	//外部输出端口Do对应的功能
	IF xSystemError OR xSystemWarning THEN
		DO_2:=FALSE;
	ELSE
		DO_2:=TRUE;
	END_IF
	DO_0:=xLED1Status;//设备运行指示灯	
	DO_1:=xLED2Status;//运行错误指示灯	
	//DO_2:= NOT xSystemError;// 机器人错误输出到外部设备
	//DO_4:=xAutoRun;//器人自动运行输出到外部设备
	
	IF CustomerPrgHandling.xWarning THEN//箱体越界信号
		WarningID:=30322;
	END_IF
	
	//////////////////////////////////////////////////////////////
	
	DeltaRobot_ErrorID:=Delta_Robot.eActiveErrorID;
	Xaxis_ErrorID	:=Axis_X.eActiveErrorID;
	Yaxis_ErrorID	:=Axis_Y.eActiveErrorID;
	Zaxis_ErrorID	:=Axis_Z.eActiveErrorID;
	A1axis_ErrorID  :=A1.eActiveErrorID;	
	A2axis_ErrorID	:=A2.eActiveErrorID;	
	A3axis_ErrorID	:=A3.eActiveErrorID;

	
	IF ErrorID<>0 THEN
		PrgOrParaErrorID:=ErrorID;
		ELSE
		PrgOrParaErrorID:=WarningID;
	END_IF

		//读取各轴的状态信息！
		ReadAxis1Info(Axis:=A1,Enable:=TRUE);
		ReadAxis2Info(Axis:=A2,Enable:=TRUE);
		ReadAxis3Info(Axis:=A3,Enable:=TRUE);

		
		//读取MCS坐标系下的位置	
		IF wstep<>20 THEN
		IF icschange=0 THEN
			AGBControl.eCoordSystem:=L_MC4P_CoordSystem.MCS;//笛卡尔坐标系MCS
			iCurrentCS:=L_MC4P_CoordSystem.MCS;
		END_IF
		IF icschange=1 THEN
			AGBControl.eCoordSystem:=L_MC4P_CoordSystem.ACS;//轴坐标系ACS
			iCurrentCS:=L_MC4P_CoordSystem.MCS;
		END_IF
		IF icschange=2 THEN
			AGBControl.eCoordSystem:=L_MC4P_CoordSystem.PCS_5;//PCS_5
			iCurrentCS:=L_MC4P_CoordSystem.PCS_5;
		END_IF
		IF icschange=4 THEN
			AGBControl.eCoordSystem:=L_MC4P_CoordSystem.PCS_6;//PCS_6
			iCurrentCS:=L_MC4P_CoordSystem.PCS_6;
		END_IF	
			ReadActPos_MCS.CoordSystem:=iCurrentCS;
			ReadActPos_MCS.Enable:=TRUE;
			ReadActPos_MCS(AxesGroup:=Delta_Robot);
			
			IF ReadActPos_MCS.Valid=TRUE THEN
				RobotPos.rRobotPosX:=LREAL_TO_REAL(ReadActPos_MCS.Position[1]);
				RobotPos.rRobotPosY:=LREAL_TO_REAL(ReadActPos_MCS.Position[2]);
				RobotPos.rRobotPosZ:=LREAL_TO_REAL(ReadActPos_MCS.Position[3]);
				
			END_IF
			
					
			ReadActPos_ACS.CoordSystem:=L_MC4P_CoordSystem.ACS;
			ReadActPos_ACS.Enable:=TRUE;
			ReadActPos_ACS(AxesGroup:=Delta_Robot);
			
			IF ReadActPos_ACS.Valid=TRUE THEN
				RobotPos.rRobotPosA1:=LREAL_TO_REAL(ReadActPos_ACS.Position[1]);
				RobotPos.rRobotPosA2:=LREAL_TO_REAL(ReadActPos_ACS.Position[2]);
				RobotPos.rRobotPosA3:=LREAL_TO_REAL(ReadActPos_ACS.Position[3]);
			END_IF
		END_IF
		
		Robot_Vel_X:=LREAL_TO_REAL(Delta_Robot.pAxis_X^.lrActVelocity);
		Robot_Vel_Y:=LREAL_TO_REAL(Delta_Robot.pAxis_Y^.lrActVelocity);
		Robot_Vel_Z:=LREAL_TO_REAL(Delta_Robot.pAxis_Z^.lrActVelocity);
		
		
		Robot_Vel_A1:=LREAL_TO_REAL(A1.lrActVelocity);
		Robot_Vel_A2:=LREAL_TO_REAL(A2.lrActVelocity);
		Robot_Vel_A3:=LREAL_TO_REAL(A3.lrActVelocity);
		//Infeed_Vel:=LREAL_TO_REAL(Infeeder.lrActVelocity);
		//Outfeed_Vel:=LREAL_TO_REAL(Outfeeder.lrActVelocity);
		//Infeed_Pos:=LREAL_TO_REAL(Infeeder.lrActPosition);
		//Outfeed_Pos:=LREAL_TO_REAL(Outfeeder.lrActPosition);
		//读取各轴的状态数据
		//读取X轴数据
		ReadXaxisPara[1].Enable:=TRUE;
		ReadXaxisPara[1].ParameterNumber:=51;
		rXaxis_PositiveLimit_Dsp:=LREAL_TO_REAL(ReadXaxisPara[1].Value);
		ReadXaxisPara[2].Enable:=TRUE;
		ReadXaxisPara[2].ParameterNumber:=52;
		rXaxis_NegativeLimit_Dsp:=LREAL_TO_REAL(ReadXaxisPara[2].Value);
		//读取Y轴数据
		ReadYaxisPara[1].Enable:=TRUE;
		ReadYaxisPara[1].ParameterNumber:=51;
		rYaxis_PositiveLimit_Dsp:=LREAL_TO_REAL(ReadYaxisPara[1].Value);
		ReadYaxisPara[2].Enable:=TRUE;
		ReadYaxisPara[2].ParameterNumber:=52;
		rYaxis_NegativeLimit_Dsp:=LREAL_TO_REAL(ReadYaxisPara[2].Value);
		//读取Z轴数据
		ReadZaxisPara[1].Enable:=TRUE;
		ReadZaxisPara[1].ParameterNumber:=51;
		rZaxis_PositiveLimit_Dsp:=LREAL_TO_REAL(ReadZaxisPara[1].Value);
		ReadZaxisPara[2].Enable:=TRUE;
		ReadZaxisPara[2].ParameterNumber:=52;
		rZaxis_NegativeLimit_Dsp:=LREAL_TO_REAL(ReadZaxisPara[2].Value);
		//读取A1轴数据
		CASE ReadA1_Step OF	
			0:
				ReadA1axisPara[1].ParameterNumber:=51;
				ReadA1axisPara[1].Enable:=TRUE;
				ReadA1_Step:=10;
			10:
				IF ReadA1axisPara[1].Valid AND NOT ReadA1axisPara[1].Error THEN
					rA1_PositiveLimit_Dsp:=LREAL_TO_REAL(ReadA1axisPara[1].Value);
					ReadA1axisPara[1].Enable:=FALSE;
					ReadA1_Step:=20;
				ELSE
					ReadA1_Step:=0;
				END_IF
			20:
				ReadA1axisPara[1].ParameterNumber:=52;
				ReadA1axisPara[1].Enable:=TRUE;
				ReadA1_Step:=30;
			30:
				IF ReadA1axisPara[1].Valid AND NOT ReadA1axisPara[1].Error THEN
					rA1_NegativeLimit_Dsp:=LREAL_TO_REAL(ReadA1axisPara[1].Value);
					ReadA1axisPara[1].Enable:=FALSE;
					ReadA1_Step:=40;
				ELSE
					ReadA1_Step:=20;
				END_IF
			40:
				ReadA1axisPara[1].ParameterNumber:=L_MC1P_IndexToParameter(16#2900,1,4);
				ReadA1axisPara[1].Enable:=TRUE;
				ReadA1_Step:=50;				
			50:
				IF ReadA1axisPara[1].Valid AND NOT ReadA1axisPara[1].Error THEN
					rA1_Vel_P1_Dsp:=LREAL_TO_REAL(ReadA1axisPara[1].Value/100000);
					ReadA1axisPara[1].Enable:=FALSE;
					ReadA1_Step:=60;
				ELSE
					ReadA1_Step:=40;
				END_IF			
			60:
				ReadA1axisPara[1].ParameterNumber:=L_MC1P_IndexToParameter(16#2900,2,2);
				ReadA1axisPara[1].Enable:=TRUE;
				ReadA1_Step:=70;
			70:
				IF ReadA1axisPara[1].Valid AND NOT ReadA1axisPara[1].Error THEN
					rA1_Vel_I1_Dsp:=LREAL_TO_REAL(ReadA1axisPara[1].Value/10);
					ReadA1axisPara[1].Enable:=FALSE;
					ReadA1_Step:=80;
				ELSE
					ReadA1_Step:=60;
				END_IF	
			80:
				ReadA1axisPara[1].ParameterNumber:=L_MC1P_IndexToParameter(16#2980,0,4);		
				ReadA1axisPara[1].Enable:=TRUE;                                                 
				ReadA1_Step:=90;                                                                
			90:                                                                                 
				IF ReadA1axisPara[1].Valid AND NOT ReadA1axisPara[1].Error THEN                 
					rA1_Pos_P1_Dsp:=LREAL_TO_REAL(ReadA1axisPara[1].Value/100);                     
					ReadA1axisPara[1].Enable:=FALSE;                                            
					ReadA1_Step:=100;                                                           
				ELSE                                                                            
					ReadA1_Step:=80;
				END_IF	
			100:
				ReadA1axisPara[1].ParameterNumber:=L_MC1P_IndexToParameter(16#6075,0,4);
				ReadA1axisPara[1].Enable:=TRUE;
				ReadA1_Step:=110;
			110:
				IF ReadA1axisPara[1].Valid AND NOT ReadA1axisPara[1].Error THEN
					rA1_Rated_Current:=LREAL_TO_REAL(ReadA1axisPara[1].Value/1000);
					ReadA1axisPara[1].Enable:=FALSE;
					ReadA1_Step:=120;
				ELSE
					ReadA1_Step:=100;
				END_IF	
			120:
				ReadA1axisPara[1].ParameterNumber:=L_MC1P_IndexToParameter(16#6078,0,4);
				ReadA1axisPara[1].Enable:=TRUE;
				ReadA1_Step:=130;
			130:
				IF ReadA1axisPara[1].Valid AND NOT ReadA1axisPara[1].Error THEN
					rA1_Actual_Current:=LREAL_TO_REAL(ReadA1axisPara[1].Value/10);
					ReadA1axisPara[1].Enable:=FALSE;
					ReadA1_Step:=140;
				ELSE
					ReadA1_Step:=120;
				END_IF	
			140:
				ReadA1axisPara[1].ParameterNumber:=L_MC1P_IndexToParameter(16#6076,0,4);
				ReadA1axisPara[1].Enable:=TRUE;
				ReadA1_Step:=150;
			150:
				IF ReadA1axisPara[1].Valid AND NOT ReadA1axisPara[1].Error THEN
					rA1_Rated_Torque:=LREAL_TO_REAL(ReadA1axisPara[1].Value/1000);
					ReadA1axisPara[1].Enable:=FALSE;
					ReadA1_Step:=160;
				ELSE
					ReadA1_Step:=140;
				END_IF	
			160:
				ReadA1axisPara[1].ParameterNumber:=L_MC1P_IndexToParameter(16#6077,0,4);
				ReadA1axisPara[1].Enable:=TRUE;
				ReadA1_Step:=170;
			170:
				IF ReadA1axisPara[1].Valid AND NOT ReadA1axisPara[1].Error THEN
					rA1_Actual_Torque:=LREAL_TO_REAL(ReadA1axisPara[1].Value/10);
					ReadA1axisPara[1].Enable:=FALSE;
					ReadA1_Step:=0;
				ELSE
					ReadA1_Step:=160;
				END_IF			
				
		END_CASE
		  
		//读取A2轴数据              
		CASE ReadA2_Step OF	
			0:
				ReadA2axisPara[1].ParameterNumber:=51;
				ReadA2axisPara[1].Enable:=TRUE;
				ReadA2_Step:=10;
			10:
				IF ReadA2axisPara[1].Valid AND NOT ReadA2axisPara[1].Error THEN
					rA2_PositiveLimit_Dsp:=LREAL_TO_REAL(ReadA2axisPara[1].Value);
					ReadA2axisPara[1].Enable:=FALSE;
					ReadA2_Step:=20;
				ELSE
					ReadA2_Step:=0;
				END_IF
			20:
				ReadA2axisPara[1].ParameterNumber:=52;
				ReadA2axisPara[1].Enable:=TRUE;
				ReadA2_Step:=30;
			30:
				IF ReadA2axisPara[1].Valid AND NOT ReadA2axisPara[1].Error THEN
					rA2_NegativeLimit_Dsp:=LREAL_TO_REAL(ReadA2axisPara[1].Value);
					ReadA2axisPara[1].Enable:=FALSE;
					ReadA2_Step:=40;
				ELSE
					ReadA2_Step:=20;
				END_IF
			40:
				ReadA2axisPara[1].ParameterNumber:=L_MC1P_IndexToParameter(16#3100,1,4);
				ReadA2axisPara[1].Enable:=TRUE;
				ReadA2_Step:=50;				
			50:
				IF ReadA2axisPara[1].Valid AND NOT ReadA2axisPara[1].Error THEN
					rA2_Vel_P1_Dsp:=LREAL_TO_REAL(ReadA2axisPara[1].Value/100000);
					ReadA2axisPara[1].Enable:=FALSE;
					ReadA2_Step:=60;
				ELSE
					ReadA2_Step:=40;
				END_IF			
			60:
				ReadA2axisPara[1].ParameterNumber:=L_MC1P_IndexToParameter(16#3100,2,2);
				ReadA2axisPara[1].Enable:=TRUE;
				ReadA2_Step:=70;
			70:
				IF ReadA2axisPara[1].Valid AND NOT ReadA2axisPara[1].Error THEN
					rA2_Vel_I1_Dsp:=LREAL_TO_REAL(ReadA2axisPara[1].Value/10);
					ReadA2axisPara[1].Enable:=FALSE;
					ReadA2_Step:=80;
				ELSE
					ReadA2_Step:=60;
				END_IF	
			80:
				ReadA2axisPara[1].ParameterNumber:=L_MC1P_IndexToParameter(16#3180,0,4);		
				ReadA2axisPara[1].Enable:=TRUE;                                                 
				ReadA2_Step:=90;                                                                
			90:                                                                                 
				IF ReadA2axisPara[1].Valid AND NOT ReadA2axisPara[1].Error THEN                 
					rA2_Pos_P1_Dsp:=LREAL_TO_REAL(ReadA2axisPara[1].Value/100);                     
					ReadA2axisPara[1].Enable:=FALSE;                                            
					ReadA2_Step:=100;                                                           
				ELSE                                                                            
					ReadA2_Step:=80;
				END_IF	
			100:
				ReadA2axisPara[1].ParameterNumber:=L_MC1P_IndexToParameter(16#6875,0,4);
				ReadA2axisPara[1].Enable:=TRUE;
				ReadA2_Step:=110;
			110:
				IF ReadA2axisPara[1].Valid AND NOT ReadA2axisPara[1].Error THEN
					rA2_Rated_Current:=LREAL_TO_REAL(ReadA2axisPara[1].Value/1000);
					ReadA2axisPara[1].Enable:=FALSE;
					ReadA2_Step:=120;
				ELSE
					ReadA2_Step:=100;
				END_IF	
			120:
				ReadA2axisPara[1].ParameterNumber:=L_MC1P_IndexToParameter(16#6878,0,4);
				ReadA2axisPara[1].Enable:=TRUE;
				ReadA2_Step:=130;
			130:
				IF ReadA2axisPara[1].Valid AND NOT ReadA2axisPara[1].Error THEN
					rA2_Actual_Current:=LREAL_TO_REAL(ReadA2axisPara[1].Value/10);
					ReadA2axisPara[1].Enable:=FALSE;
					ReadA2_Step:=140;
				ELSE
					ReadA2_Step:=120;
				END_IF	
			140:
				ReadA2axisPara[1].ParameterNumber:=L_MC1P_IndexToParameter(16#6876,0,4);
				ReadA2axisPara[1].Enable:=TRUE;
				ReadA2_Step:=150;
			150:
				IF ReadA2axisPara[1].Valid AND NOT ReadA2axisPara[1].Error THEN
					rA2_Rated_Torque:=LREAL_TO_REAL(ReadA2axisPara[1].Value/1000);
					ReadA2axisPara[1].Enable:=FALSE;
					ReadA2_Step:=160;
				ELSE
					ReadA2_Step:=140;
				END_IF	
			160:
				ReadA2axisPara[1].ParameterNumber:=L_MC1P_IndexToParameter(16#6877,0,4);
				ReadA2axisPara[1].Enable:=TRUE;
				ReadA2_Step:=170;
			170:
				IF ReadA2axisPara[1].Valid AND NOT ReadA2axisPara[1].Error THEN
					rA2_Actual_Torque:=LREAL_TO_REAL(ReadA2axisPara[1].Value/10);
					ReadA2axisPara[1].Enable:=FALSE;
					ReadA2_Step:=0;
				ELSE
					ReadA2_Step:=160;
				END_IF			
				
		END_CASE
		

		//读取A3轴数据
		CASE ReadA3_Step OF	
			0:
				ReadA3axisPara[1].ParameterNumber:=51;
				ReadA3axisPara[1].Enable:=TRUE;
				ReadA3_Step:=10;
			10:
				IF ReadA3axisPara[1].Valid AND NOT ReadA3axisPara[1].Error THEN
					rA3_PositiveLimit_Dsp:=LREAL_TO_REAL(ReadA3axisPara[1].Value);
					ReadA3axisPara[1].Enable:=FALSE;
					ReadA3_Step:=20;
				ELSE
					ReadA3_Step:=0;
				END_IF
			20:
				ReadA3axisPara[1].ParameterNumber:=52;
				ReadA3axisPara[1].Enable:=TRUE;
				ReadA3_Step:=30;
			30:
				IF ReadA3axisPara[1].Valid AND NOT ReadA3axisPara[1].Error THEN
					rA3_NegativeLimit_Dsp:=LREAL_TO_REAL(ReadA3axisPara[1].Value);
					ReadA3axisPara[1].Enable:=FALSE;
					ReadA3_Step:=40;
				ELSE
					ReadA3_Step:=20;
				END_IF
			40:
				ReadA3axisPara[1].ParameterNumber:=L_MC1P_IndexToParameter(16#2900,1,4);
				ReadA3axisPara[1].Enable:=TRUE;
				ReadA3_Step:=50;				
			50:
				IF ReadA3axisPara[1].Valid AND NOT ReadA3axisPara[1].Error THEN
					rA3_Vel_P1_Dsp:=LREAL_TO_REAL(ReadA3axisPara[1].Value/100000);
					ReadA3axisPara[1].Enable:=FALSE;
					ReadA3_Step:=60;
				ELSE
					ReadA3_Step:=40;
				END_IF			
			60:
				ReadA3axisPara[1].ParameterNumber:=L_MC1P_IndexToParameter(16#2900,2,2);
				ReadA3axisPara[1].Enable:=TRUE;
				ReadA3_Step:=70;
			70:
				IF ReadA3axisPara[1].Valid AND NOT ReadA3axisPara[1].Error THEN
					rA3_Vel_I1_Dsp:=LREAL_TO_REAL(ReadA3axisPara[1].Value/10);
					ReadA3axisPara[1].Enable:=FALSE;
					ReadA3_Step:=80;
				ELSE
					ReadA3_Step:=60;
				END_IF	
			80:
				ReadA3axisPara[1].ParameterNumber:=L_MC1P_IndexToParameter(16#2980,0,4);		
				ReadA3axisPara[1].Enable:=TRUE;                                                 
				ReadA3_Step:=90;                                                                
			90:                                                                                 
				IF ReadA3axisPara[1].Valid AND NOT ReadA3axisPara[1].Error THEN                 
					rA3_Pos_P1_Dsp:=LREAL_TO_REAL(ReadA3axisPara[1].Value/100);                     
					ReadA3axisPara[1].Enable:=FALSE;                                            
					ReadA3_Step:=100;                                                           
				ELSE                                                                            
					ReadA3_Step:=80;
				END_IF	
			100:
				ReadA3axisPara[1].ParameterNumber:=L_MC1P_IndexToParameter(16#6075,0,4);
				ReadA3axisPara[1].Enable:=TRUE;
				ReadA3_Step:=110;
			110:
				IF ReadA3axisPara[1].Valid AND NOT ReadA3axisPara[1].Error THEN
					rA3_Rated_Current:=LREAL_TO_REAL(ReadA3axisPara[1].Value/1000);
					ReadA3axisPara[1].Enable:=FALSE;
					ReadA3_Step:=120;
				ELSE
					ReadA3_Step:=100;
				END_IF	
			120:
				ReadA3axisPara[1].ParameterNumber:=L_MC1P_IndexToParameter(16#6078,0,4);
				ReadA3axisPara[1].Enable:=TRUE;
				ReadA3_Step:=130;
			130:
				IF ReadA3axisPara[1].Valid AND NOT ReadA3axisPara[1].Error THEN
					rA3_Actual_Current:=LREAL_TO_REAL(ReadA3axisPara[1].Value/10);
					ReadA3axisPara[1].Enable:=FALSE;
					ReadA3_Step:=140;
				ELSE
					ReadA3_Step:=120;
				END_IF	
			140:
				ReadA3axisPara[1].ParameterNumber:=L_MC1P_IndexToParameter(16#6076,0,4);
				ReadA3axisPara[1].Enable:=TRUE;
				ReadA3_Step:=150;
			150:
				IF ReadA3axisPara[1].Valid AND NOT ReadA3axisPara[1].Error THEN
					rA3_Rated_Torque:=LREAL_TO_REAL(ReadA3axisPara[1].Value/1000);
					ReadA3axisPara[1].Enable:=FALSE;
					ReadA3_Step:=160;
				ELSE
					ReadA3_Step:=140;
				END_IF	
			160:
				ReadA3axisPara[1].ParameterNumber:=L_MC1P_IndexToParameter(16#6077,0,4);
				ReadA3axisPara[1].Enable:=TRUE;
				ReadA3_Step:=170;
			170:
				IF ReadA3axisPara[1].Valid AND NOT ReadA3axisPara[1].Error THEN
					rA3_Actual_Torque:=LREAL_TO_REAL(ReadA3axisPara[1].Value/10);
					ReadA3axisPara[1].Enable:=FALSE;
					ReadA3_Step:=0;
				ELSE
					ReadA3_Step:=160;
				END_IF			
				
		END_CASE  
		
		//读取AuxC轴数据
		CASE ReadAuxC_Step OF	
			0:
				ReadAuxCaxisPara[1].ParameterNumber:=51;
				ReadAuxCaxisPara[1].Enable:=TRUE;
				ReadAuxC_Step:=10;
			10:
				IF ReadAuxCaxisPara[1].Valid AND NOT ReadAuxCaxisPara[1].Error THEN
					rAuxC_PositiveLimit_Dsp:=LREAL_TO_REAL(ReadAuxCaxisPara[1].Value);
					ReadAuxCaxisPara[1].Enable:=FALSE;
					ReadAuxC_Step:=20;
				ELSE
					ReadAuxC_Step:=0;
				END_IF
			20:
				ReadAuxCaxisPara[1].ParameterNumber:=52;
				ReadAuxCaxisPara[1].Enable:=TRUE;
				ReadAuxC_Step:=30;
			30:
				IF ReadAuxCaxisPara[1].Valid AND NOT ReadAuxCaxisPara[1].Error THEN
					rAuxC_NegativeLimit_Dsp:=LREAL_TO_REAL(ReadAuxCaxisPara[1].Value);
					ReadAuxCaxisPara[1].Enable:=FALSE;
					ReadAuxC_Step:=40;
				ELSE
					ReadAuxC_Step:=20;
				END_IF
			40:
				ReadAuxCaxisPara[1].ParameterNumber:=L_MC1P_IndexToParameter(16#3100,1,4);
				ReadAuxCaxisPara[1].Enable:=TRUE;
				ReadAuxC_Step:=50;				
			50:
				IF ReadAuxCaxisPara[1].Valid AND NOT ReadAuxCaxisPara[1].Error THEN
					rAuxC_Vel_P1_Dsp:=LREAL_TO_REAL(ReadAuxCaxisPara[1].Value/100000);
					ReadAuxCaxisPara[1].Enable:=FALSE;
					ReadAuxC_Step:=60;
				ELSE
					ReadAuxC_Step:=40;
				END_IF			
			60:
				ReadAuxCaxisPara[1].ParameterNumber:=L_MC1P_IndexToParameter(16#3100,2,2);
				ReadAuxCaxisPara[1].Enable:=TRUE;
				ReadAuxC_Step:=70;
			70:
				IF ReadAuxCaxisPara[1].Valid AND NOT ReadAuxCaxisPara[1].Error THEN
					rAuxC_Vel_I1_Dsp:=LREAL_TO_REAL(ReadAuxCaxisPara[1].Value/10);
					ReadAuxCaxisPara[1].Enable:=FALSE;
					ReadAuxC_Step:=80;
				ELSE
					ReadAuxC_Step:=60;
				END_IF	
			80:
				ReadAuxCaxisPara[1].ParameterNumber:=L_MC1P_IndexToParameter(16#3180,0,4);		
				ReadAuxCaxisPara[1].Enable:=TRUE;                                                 
				ReadAuxC_Step:=90;                                                                
			90:                                                                                 
				IF ReadAuxCaxisPara[1].Valid AND NOT ReadAuxCaxisPara[1].Error THEN                 
					rAuxC_Pos_P1_Dsp:=LREAL_TO_REAL(ReadAuxCaxisPara[1].Value/100);                     
					ReadAuxCaxisPara[1].Enable:=FALSE;                                            
					ReadAuxC_Step:=100;                                                           
				ELSE                                                                            
					ReadAuxC_Step:=80;
				END_IF	
			100:
				ReadAuxCaxisPara[1].ParameterNumber:=L_MC1P_IndexToParameter(16#6875,0,4);
				ReadAuxCaxisPara[1].Enable:=TRUE;
				ReadAuxC_Step:=110;
			110:
				IF ReadAuxCaxisPara[1].Valid AND NOT ReadAuxCaxisPara[1].Error THEN
					rAuxC_Rated_Current:=LREAL_TO_REAL(ReadAuxCaxisPara[1].Value/1000);
					ReadAuxCaxisPara[1].Enable:=FALSE;
					ReadAuxC_Step:=120;
				ELSE
					ReadAuxC_Step:=100;
				END_IF	
			120:
				ReadAuxCaxisPara[1].ParameterNumber:=L_MC1P_IndexToParameter(16#6878,0,4);
				ReadAuxCaxisPara[1].Enable:=TRUE;
				ReadAuxC_Step:=130;
			130:
				IF ReadAuxCaxisPara[1].Valid AND NOT ReadAuxCaxisPara[1].Error THEN
					rAuxC_Actual_Current:=LREAL_TO_REAL(ReadAuxCaxisPara[1].Value/10);
					ReadAuxCaxisPara[1].Enable:=FALSE;
					ReadAuxC_Step:=140;
				ELSE
					ReadAuxC_Step:=120;
				END_IF	
			140:
				ReadAuxCaxisPara[1].ParameterNumber:=L_MC1P_IndexToParameter(16#6876,0,4);
				ReadAuxCaxisPara[1].Enable:=TRUE;
				ReadAuxC_Step:=150;
			150:
				IF ReadAuxCaxisPara[1].Valid AND NOT ReadAuxCaxisPara[1].Error THEN
					rAuxC_Rated_Torque:=LREAL_TO_REAL(ReadAuxCaxisPara[1].Value/1000);
					ReadAuxCaxisPara[1].Enable:=FALSE;
					ReadAuxC_Step:=160;
				ELSE
					ReadAuxC_Step:=140;
				END_IF	
			160:
				ReadAuxCaxisPara[1].ParameterNumber:=L_MC1P_IndexToParameter(16#6877,0,4);
				ReadAuxCaxisPara[1].Enable:=TRUE;
				ReadAuxC_Step:=170;
			170:
				IF ReadAuxCaxisPara[1].Valid AND NOT ReadAuxCaxisPara[1].Error THEN
					rAuxC_Actual_Torque:=LREAL_TO_REAL(ReadAuxCaxisPara[1].Value/10);
					ReadAuxCaxisPara[1].Enable:=FALSE;
					ReadAuxC_Step:=0;
				ELSE
					ReadAuxC_Step:=160;
				END_IF			
				
		END_CASE
		//读取Infeeder轴数据                                             
		 ReadInfeederPara.xEnable:=TRUE;
		 xInfeederDirectionDsp:=ReadInfeederPara.xOrientation;		
		 //rInfeederPosResolutionDsp:=DWORD_TO_REAL(ReadInfeederPara.dwPosResolution);		
		 //rInfeederGearRedRatioDsp:=DWORD_TO_REAL(ReadInfeederPara.dwGearNumerator)/DWORD_TO_REAL(ReadInfeederPara.dwGearDenominator);		
		 rInfeederFeedConstDsp:=LREAL_TO_REAL(ReadInfeederPara.lrFeedconstant);			
		 //rInfeederCycleLengthDsp:=LREAL_TO_REAL(ReadInfeederPara.lrCycleLength);		
		 
		//读取Outfeeder轴数据
		ReadOutfeederPara.xEnable:=TRUE;
		xOutfeederDirectionDsp:=ReadOutfeederPara.xOrientation;		
		//rOutfeederPosResolutionDsp:=DWORD_TO_REAL(ReadOutfeederPara.dwPosResolution);		
		//rOutfeederGearRedRatioDsp:=DWORD_TO_REAL(ReadOutfeederPara.dwGearNumerator)/DWORD_TO_REAL(ReadOutfeederPara.dwGearDenominator);		
		rOutfeederFeedConstDsp:=LREAL_TO_REAL(ReadOutfeederPara.lrFeedconstant);			
		//rOutfeederCycleLengthDsp:=LREAL_TO_REAL(ReadOutfeederPara.lrCycleLength);
		
				rInfeederPosResolutionDsp:=rInfeederPosResolution;
				rInfeederGearRedRatioDsp:=rInfeederGearRedRatio;
				rOutfeederPosResolutionDsp:=rOutfeederPosResolution;
				rOutfeederGearRedRatioDsp:=rOutfeederGearRedRatio;
				
	ReadXaxisPara[1](Axis:=Axis_X); ReadXaxisPara[2](Axis:=Axis_X);	
	ReadYaxisPara[1](Axis:=Axis_Y); ReadYaxisPara[2](Axis:=Axis_Y);		
	ReadZaxisPara[1](Axis:=Axis_Z); ReadZaxisPara[2](Axis:=Axis_Z);
	
	ReadA1axisPara[1](Axis:=A1);	
	ReadA2axisPara[1](Axis:=A2); 
	ReadA3axisPara[1](Axis:=A3); 
 
	//ReadInfeederPara(Axis:=Infeeder);
	//ReadOutfeederPara(Axis:=Outfeeder);
END_ACTION

ACTION A10_CameraInterface:

END_ACTION

ACTION A01_EditPrg:
IF NOT xAutoRun AND xMainInit THEN	
	CustomerPrgEdit(axSavePrgNo:=p_axSavePrgNo,adr_iCurrentPrgNum:=p_iCurrentPrgNum,xSaveRunPra:=xSaveRunPra,
		rFollowBias_X:=rFollowBias_X,rFollowBias_Y:=rFollowBias_Y,rSuckerDropHeight:=rSuckerDropHeight,
		rBelt1_ClutchPra:=rBelt1_ClutchPra,rBelt2_ClutchPra:=rBelt2_ClutchPra,
		rSuck_Gas_OpenTime:=rSuck_Gas_OpenTime,rBlow_Gas_OpenTime:=rBlow_Gas_OpenTime,rBlowGasTime:=rBlowGasTime,
		iBox_ExceptionDeal:=iBox_ExceptionDeal,		
		iSelfadaptPickSwitch:=iSelfadaptPickSwitch,
		rPnPDurationNegativeLimit:=rPnPDurationNegative,
	    rPnPDurationPositiveLimit:=rPnPDurationPositive,
		iProdDeformation:=iProdDeformation,
		CustomerPrg:=CustomerPrg,aLRPP_TeachPoints:=aLRPP_TeachPoints);
END_IF
END_ACTION

ACTION A10_Homing:
IF  NOT xAutoRun AND xMainInit  THEN	
		/////////////////////1.设定各轴零位					
	L_McSetPosition[1](
		Axis		:= A1, 
		Execute		:= xSetA1Position, 
		Position	:=rA1SetHomePostion , 
		Relative	:= , 
		ExecutionMode:= , 
		Done=> , 
		Busy=> , 
		Error=> , 
		ErrorID=> );
	
	L_McSetPosition[2](
		Axis:= A2, 
		Execute:= xSetA2Position , 
		Position:=rA2SetHomePostion  , 
		Relative:= , 
		ExecutionMode:= , 
		Done=> , 
		Busy=> , 
		Error=> , 
		ErrorID=> );
	
	L_McSetPosition[3](
		Axis:= A3, 
		Execute:= xSetA3Position , 
		Position:=rA3SetHomePostion  , 
		Relative:= , 
		ExecutionMode:= , 
		Done=> , 
		Busy=> , 
		Error=> , 
		ErrorID=> );			
		
	IF	L_McSetPosition[1].Done=TRUE THEN
		xSetA1Position:=FALSE;
	END_IF
	
	IF	L_McSetPosition[2].Done=TRUE THEN
		xSetA2Position:=FALSE;
	END_IF
	
	IF	L_McSetPosition[3].Done=TRUE THEN
		xSetA3Position:=FALSE;
	END_IF
	

END_IF
END_ACTION

ACTION A50_Brake:

IF NOT xAutoRun AND xMainInit THEN	
	// A1 Brake Open
	
	A1_BrakeDelay(IN:=BYTE_TO_BOOL(bA1_Open), PT:=T#2S , Q=> , ET=> );		
	
	A1_BrakeControl(
		Axis:=A1 , 
		xEnable:=A1_BrakeDelay.Q  , 
		xReleaseBrake:=BYTE_TO_BOOL(bA1_Open) AND (NOT AGBControl.xAxesGroupEnabled) , 
		lrTorqueAdd:= , 
		xValid=> , 
		xBusy=> , 
		xError=> , 
		eErrorID=> , 
		xBrakeReleaseOut=> , 
		xBrakeReleased=>xA1_BrakeOpenStatus , 
		lrActTorque=> );
	
	bA1_BrakeOpenStatus:=BOOL_TO_BYTE(xA1_BrakeOpenStatus);
	
	// A2 Brake Open
	A2_BrakeDelay(IN:=BYTE_TO_BOOL(bA2_Open), PT:=T#2S , Q=> , ET=> );	
	A2_BrakeControl(
		Axis:=A2 , 
		xEnable:=A2_BrakeDelay.Q , 
		xReleaseBrake:=BYTE_TO_BOOL(bA2_Open) AND (NOT AGBControl.xAxesGroupEnabled)  , 
		lrTorqueAdd:= , 
		xValid=> , 
		xBusy=> , 
		xError=> , 
		eErrorID=> , 
		xBrakeReleaseOut=> , 
		xBrakeReleased=>xA2_BrakeOpenStatus, 
		lrActTorque=> );
	
	bA2_BrakeOpenStatus:=BOOL_TO_BYTE(xA2_BrakeOpenStatus);
	
	// A3 Brake Open
	A3_BrakeDelay(IN:=BYTE_TO_BOOL(bA3_Open), PT:=T#2S , Q=> , ET=> );	
	A3_BrakeControl(
		Axis:=A3 , 
		xEnable:=A3_BrakeDelay.Q , 
		xReleaseBrake:=BYTE_TO_BOOL(bA3_Open) AND (NOT AGBControl.xAxesGroupEnabled)  , 
		lrTorqueAdd:= , 
		xValid=> , 
		xBusy=> , 
		xError=> , 
		eErrorID=> , 
		xBrakeReleaseOut=> , 
		xBrakeReleased=>xA3_BrakeOpenStatus, 
		lrActTorque=> );
	
	bA3_BrakeOpenStatus:=BOOL_TO_BYTE(xA3_BrakeOpenStatus);
	
	// AuxC Brake Open

END_IF
END_ACTION

END_PROGRAM

// Controller_3200C/Application/FunctionBlock/_L_MC1B_PackBytesToDWord
FUNCTION _L_MC1B_PackBytesToDWord : DWORD
VAR_INPUT

	pPointerToByte	: POINTER TO BYTE;
	iNumOfByte		: INT;	
END_VAR
VAR
	dwNumber : DWORD;
	wNumber : WORD;
	pPointerToByte2	: POINTER TO  ARRAY[0..1] OF BYTE;
	pPointerToByte4	: POINTER TO  ARRAY[0..3] OF BYTE;

END_VAR

IF pPointerToByte = 0 
OR iNumOfByte < 1
OR iNumOfByte > 4
THEN
	RETURN;
END_IF



CASE iNumOfByte OF 
	1:
	pPointerToByte2 := pPointerToByte;	
	wNumber := MEM.PackBytesToWord(
						byLowByte 	:=pPointerToByte^, 
						byHighByte	:= 0);
	
	_L_MC1B_PackBytesToDword := WORD_TO_DWORD(wNumber);
	2:
	pPointerToByte2 := pPointerToByte;	
	wNumber := MEM.PackBytesToWord(
						byHighByte	:=pPointerToByte2^[1], 
						byLowByte	:= pPointerToByte2^[0]);
	
	_L_MC1B_PackBytesToDword := WORD_TO_DWORD(wNumber);
	3:
	pPointerToByte4 := pPointerToByte;
	
	dwNumber := MEM.PackBytesToDword(
		byHHByte:=  0,
		byHLByte:= pPointerToByte4^[2],
		byLHByte:= pPointerToByte4^[1], 
		byLLByte:= pPointerToByte4^[0], );
	
	_L_MC1B_PackBytesToDword := (dwNumber);
	
	4:
	pPointerToByte4 := pPointerToByte;
	
	dwNumber := MEM.PackBytesToDword(
		byHHByte:= pPointerToByte4^[3], 
		byHLByte:= pPointerToByte4^[2], 
		byLHByte:= pPointerToByte4^[1], 
		byLLByte:= pPointerToByte4^[0]);
	
	_L_MC1B_PackBytesToDword := (dwNumber);
	
END_CASE

END_FUNCTION

// Controller_3200C/Application/FunctionBlock/_L_MC1B_PackBytesToLreal
FUNCTION _L_MC1B_PackBytesToLreal : LREAL
VAR_INPUT

	pPointerToByte	: POINTER TO BYTE;
	iNumOfByte		: INT;	
END_VAR
VAR
	dwNumber : DWORD;
	wNumber : WORD;
	pPointerToByte2	: POINTER TO  ARRAY[0..1] OF BYTE;
	pPointerToByte4	: POINTER TO  ARRAY[0..3] OF BYTE;

END_VAR

IF pPointerToByte = 0 
OR iNumOfByte < 1
OR iNumOfByte > 4
THEN
	RETURN;
END_IF



CASE iNumOfByte OF 
	1:
	pPointerToByte2 := pPointerToByte;	
	IF 	(pPointerToByte2^[0] AND 2#1000_0000)  = 0  THEN
	wNumber := MEM.PackBytesToWord(
						byLowByte 	:=pPointerToByte^, 
						byHighByte	:= 0);
	
	_L_MC1B_PackBytesToLreal := WORD_TO_LREAL(wNumber);
	  
	ELSE
		wNumber := MEM.PackBytesToWord(
						byHighByte	:=0, 
						byLowByte	:=pPointerToByte^,);
		_L_MC1B_PackBytesToLreal :=  WORD_TO_LREAL(wNumber)- 256;
		
	END_IF

	2:
		
	pPointerToByte2 := pPointerToByte;	
	IF 	(pPointerToByte2^[1] AND 2#1000_0000)  = 0  THEN
	wNumber := MEM.PackBytesToWord(
						byHighByte	:=pPointerToByte2^[1], 
						byLowByte	:= pPointerToByte2^[0]);
	
	_L_MC1B_PackBytesToLreal := WORD_TO_LREAL(wNumber);
	
	ELSE
		wNumber := MEM.PackBytesToWord(
						byHighByte	:=pPointerToByte2^[1], 
						byLowByte	:= pPointerToByte2^[0]);
		_L_MC1B_PackBytesToLreal :=  WORD_TO_LREAL(wNumber)- 65536;
		
	END_IF
	
	
	3:
	
	pPointerToByte4 := pPointerToByte;
	
	IF 	(pPointerToByte4^[2] AND 2#1000_0000)  = 0  THEN
	dwNumber := MEM.PackBytesToDword(
		byHHByte:=  0,
		byHLByte:= pPointerToByte4^[2],
		byLHByte:= pPointerToByte4^[1], 
		byLLByte:= pPointerToByte4^[0], );

	_L_MC1B_PackBytesToLreal := DWORD_TO_LREAL(dwNumber);
	
	    ELSE
		dwNumber := MEM.PackBytesToDword(
		byHHByte:=  0,
		byHLByte:= pPointerToByte4^[2], 
		byLHByte:= pPointerToByte4^[1], 
		byLLByte:= pPointerToByte4^[0]);
		_L_MC1B_PackBytesToLreal :=  DWORD_TO_LREAL(dwNumber)- 16777216;
		
	END_IF
	
	4:
	pPointerToByte4 := pPointerToByte;
	

	IF 	(pPointerToByte4^[3] AND 2#1000_0000)  = 0  THEN
		
		dwNumber := MEM.PackBytesToDword(
		byHHByte:= pPointerToByte4^[3], 
		byHLByte:= pPointerToByte4^[2], 
		byLHByte:= pPointerToByte4^[1], 
		byLLByte:= pPointerToByte4^[0]);
		_L_MC1B_PackBytesToLreal := DWORD_TO_LREAL(dwNumber);
		
    ELSE
		dwNumber := MEM.PackBytesToDword(
		byHHByte:= pPointerToByte4^[3] , 
		byHLByte:= pPointerToByte4^[2], 
		byLHByte:= pPointerToByte4^[1], 
		byLLByte:= pPointerToByte4^[0]);
		_L_MC1B_PackBytesToLreal :=  DWORD_TO_LREAL(dwNumber)- 4294967296;
		
	END_IF
		
(*	1:
	pPointerToByte2 := pPointerToByte;	
	wNumber := MEM.PackBytesToWord(
						byLowByte 	:=pPointerToByte^, 
						byHighByte	:= 0);
	
	_L_MC1B_PackBytesToLreal := WORD_TO_LREAL(wNumber);
	2:
	pPointerToByte2 := pPointerToByte;	
	wNumber := MEM.PackBytesToWord(
						byHighByte	:=pPointerToByte2^[1], 
						byLowByte	:= pPointerToByte2^[0]);
	
	_L_MC1B_PackBytesToLreal := WORD_TO_LREAL(wNumber);
	3:
	pPointerToByte4 := pPointerToByte;
	
	dwNumber := MEM.PackBytesToDword(
		byHHByte:=  0,
		byHLByte:= pPointerToByte4^[2],
		byLHByte:= pPointerToByte4^[1], 
		byLLByte:= pPointerToByte4^[0], );
	
	_L_MC1B_PackBytesToLreal := DWORD_TO_LREAL(dwNumber);
	
	4:
	pPointerToByte4 := pPointerToByte;
	
	dwNumber := MEM.PackBytesToDword(
		byHHByte:= pPointerToByte4^[3], 
		byHLByte:= pPointerToByte4^[2], 
		byLHByte:= pPointerToByte4^[1], 
		byLLByte:= pPointerToByte4^[0]);
	
	_L_MC1B_PackBytesToLreal := DWORD_TO_LREAL(dwNumber);
*)	
END_CASE

END_FUNCTION

// Controller_3200C/Application/FunctionBlock/_L_MC1B_PackBytesToWord
FUNCTION _L_MC1B_PackBytesToWord : WORD
VAR_INPUT

	pPointerToByte	: POINTER TO BYTE;
	iNumOfByte		: INT;	
END_VAR
VAR
	dwNumber : DWORD;
	wNumber : WORD;
	pPointerToByte2	: POINTER TO  ARRAY[0..1] OF BYTE;
	pPointerToByte4	: POINTER TO  ARRAY[0..3] OF BYTE;

END_VAR

IF pPointerToByte = 0 
OR iNumOfByte < 1
OR iNumOfByte > 4
THEN
	RETURN;
END_IF



CASE iNumOfByte OF 
	1:
	pPointerToByte2 := pPointerToByte;	
	wNumber := MEM.PackBytesToWord(
						byLowByte 	:=pPointerToByte^, 
						byHighByte	:= 0);
	
	_L_MC1B_PackBytesToWord := (wNumber);
	2:
	pPointerToByte2 := pPointerToByte;	
	wNumber := MEM.PackBytesToWord(
						byHighByte	:=pPointerToByte2^[1], 
						byLowByte	:= pPointerToByte2^[0]);
	
	_L_MC1B_PackBytesToWord := (wNumber);
	3:
	pPointerToByte4 := pPointerToByte;
	
	dwNumber := MEM.PackBytesToDword(
		byHHByte:=  0,
		byHLByte:= pPointerToByte4^[2],
		byLHByte:= pPointerToByte4^[1], 
		byLLByte:= pPointerToByte4^[0], );
	
	_L_MC1B_PackBytesToWord := DWORD_TO_WORD(dwNumber);
	
	4:
	pPointerToByte4 := pPointerToByte;
	
	dwNumber := MEM.PackBytesToDword(
		byHHByte:= pPointerToByte4^[3], 
		byHLByte:= pPointerToByte4^[2], 
		byLHByte:= pPointerToByte4^[1], 
		byLLByte:= pPointerToByte4^[0]);
	
	_L_MC1B_PackBytesToWord := DWORD_TO_WORD(dwNumber);
	
END_CASE

END_FUNCTION

// Controller_3200C/Application/FunctionBlock/_L_MC1B_PackDWordToByte
FUNCTION _L_MC1B_PackDWordToByte 
VAR_INPUT
	dwValue			: DWORD;
	pPointerToByte	: POINTER TO BYTE;
	iNumOfByte		: INT;	
END_VAR
VAR

	wNumber : WORD;
	pPointerToByte2	: POINTER TO  ARRAY[0..1] OF BYTE;
	pPointerToByte3	: POINTER TO  ARRAY[0..2] OF BYTE;
	pPointerToByte4	: POINTER TO  ARRAY[0..3] OF BYTE;

	UnpackWord1 : MEM.UnpackWord;
	UnpackDWord1: MEM.UnpackDWord;
END_VAR

IF pPointerToByte = 0 
OR iNumOfByte < 1
OR iNumOfByte > 4
THEN
	RETURN;
END_IF


CASE iNumOfByte OF 
	1:
	wNumber 		:= DWORD_TO_WORD(dwValue);
	 UnpackWord1(
						wValue 		:= wNumber,							
						byLowByte	=> pPointerToByte^ 
						);
						
						
	2:
	pPointerToByte2 := pPointerToByte;	
	wNumber 		:= DWORD_TO_WORD(dwValue);
	UnpackWord1(
						wValue 		:= wNumber,							
						byHighByte	=> pPointerToByte2^[1], 
						byLowByte	=> pPointerToByte2^[0]);

						
						

	3:
	pPointerToByte3 := pPointerToByte;

	UnpackDWord1(
		dwValue 		:= dwValue,		
			//byHHByte 	=> 0, 
			byHLByte 	=> pPointerToByte3^[2], 
			byLHByte 	=> pPointerToByte3^[1], 
			byLLByte 	=> pPointerToByte3^[0]
			);
	

	
	4:
	pPointerToByte4 := pPointerToByte;
	UnpackDWord1(
			dwValue  	:= dwValue,
			byHHByte 	=> pPointerToByte4^[3], 
			byHLByte 	=> pPointerToByte4^[2], 
			byLHByte 	=> pPointerToByte4^[1], 
			byLLByte 	=> pPointerToByte4^[0]
							 );
	
	
END_CASE

END_FUNCTION

// Controller_3200C/Application/FunctionBlock/_L_MC1B_PackLRealToByte
FUNCTION _L_MC1B_PackLRealToByte 
VAR_INPUT
	lrValue			: LREAL;
	pPointerToByte	: POINTER TO BYTE;
	iNumOfByte		: INT;	
END_VAR
VAR

	dwNumber : DWORD;
	wNumber : WORD;
	pPointerToByte2	: POINTER TO  ARRAY[0..1] OF BYTE;
	pPointerToByte3	: POINTER TO  ARRAY[0..2] OF BYTE;
	pPointerToByte4	: POINTER TO  ARRAY[0..3] OF BYTE;

	UnpackWord1 : MEM.UnpackWord;
	UnpackDWord1: MEM.UnpackDWord;
END_VAR

IF pPointerToByte = 0 
OR iNumOfByte < 1
OR iNumOfByte > 4
THEN
	RETURN;
END_IF


CASE iNumOfByte OF 
	1:
	wNumber 		:= LREAL_TO_WORD(lrValue);
	 UnpackWord1(
						wValue 		:= wNumber,							
						byLowByte	=> pPointerToByte^ 
						);
						
						
	2:
	pPointerToByte2 := pPointerToByte;	
	wNumber 		:= LREAL_TO_WORD(lrValue);
	UnpackWord1(
						wValue 		:= wNumber,							
						byHighByte	=> pPointerToByte2^[1], 
						byLowByte	=> pPointerToByte2^[0]);

						
						

	3:
	pPointerToByte3 := pPointerToByte;
	dwNumber 		:= LREAL_TO_DWORD(lrValue);
	UnpackDWord1(
		dwValue 		:= dwNumber,		
			//byHHByte 	=> 0, 
			byHLByte 	=> pPointerToByte3^[2], 
			byLHByte 	=> pPointerToByte3^[1], 
			byLLByte 	=> pPointerToByte3^[0]
			);
	

	
	4:
	pPointerToByte4 := pPointerToByte;
	dwNumber 		:= LREAL_TO_DWORD(lrValue);
	UnpackDWord1(
			dwValue  	:= dwNumber,
			byHHByte 	=> pPointerToByte4^[3], 
			byHLByte 	=> pPointerToByte4^[2], 
			byLHByte 	=> pPointerToByte4^[1], 
			byLLByte 	=> pPointerToByte4^[0]
							 );
	
	
END_CASE

END_FUNCTION

// Controller_3200C/Application/FunctionBlock/_L_MC1B_PackWordToByte
FUNCTION _L_MC1B_PackWordToByte 
VAR_INPUT
	wValue			: WORD;
	pPointerToByte	: POINTER TO BYTE;
	iNumOfByte		: INT;	
END_VAR
VAR
	pPointerToByte2	: POINTER TO  ARRAY[0..1] OF BYTE;
	UnpackWord1 : MEM.UnpackWord;
END_VAR

IF pPointerToByte = 0 
OR iNumOfByte < 1
OR iNumOfByte > 4
THEN
	RETURN;
END_IF


CASE iNumOfByte OF 
	1:

	 UnpackWord1(
						wValue 		:= wValue,							
						byLowByte	=> pPointerToByte^ 
						);
						
						
	2,3,4:
	pPointerToByte2 := pPointerToByte;	
	UnpackWord1(
						wValue 		:= wValue,							
						byHighByte	=> pPointerToByte2^[1], 
						byLowByte	=> pPointerToByte2^[0]);

						
						

	
	
	
END_CASE

END_FUNCTION

// Controller_3200C/Application/B5_VISUAL/DeltaRobot
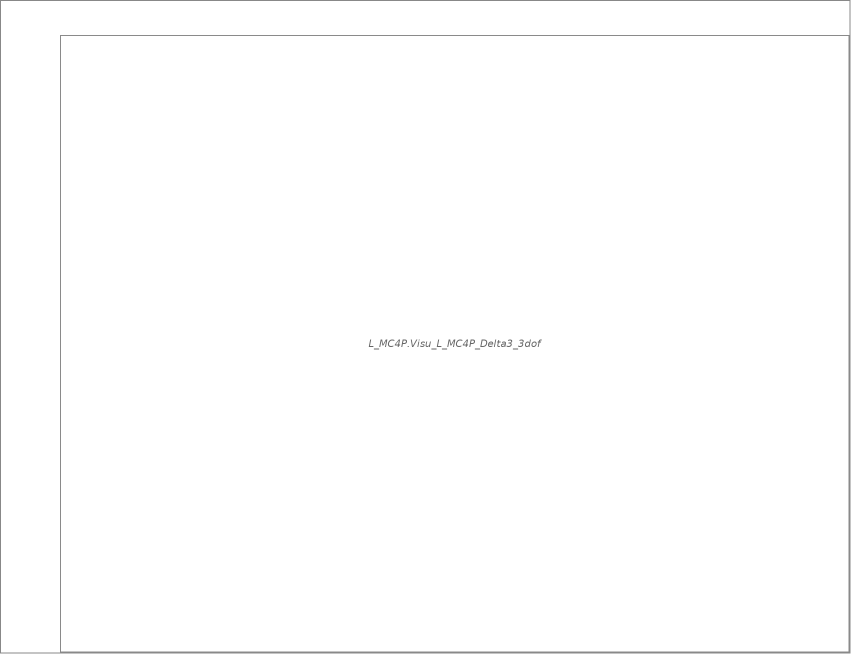
VISUALIZATION DeltaRobot  // 851x654
    Frame (60,35 789x617)
        shows L_MC4P.Visu_L_MC4P_Delta3_3dof(m_Input_AxesGroupRef := Delta_Robot)
END_VISUALIZATION

// Controller_3200C/Application/B5_VISUAL/ABControl
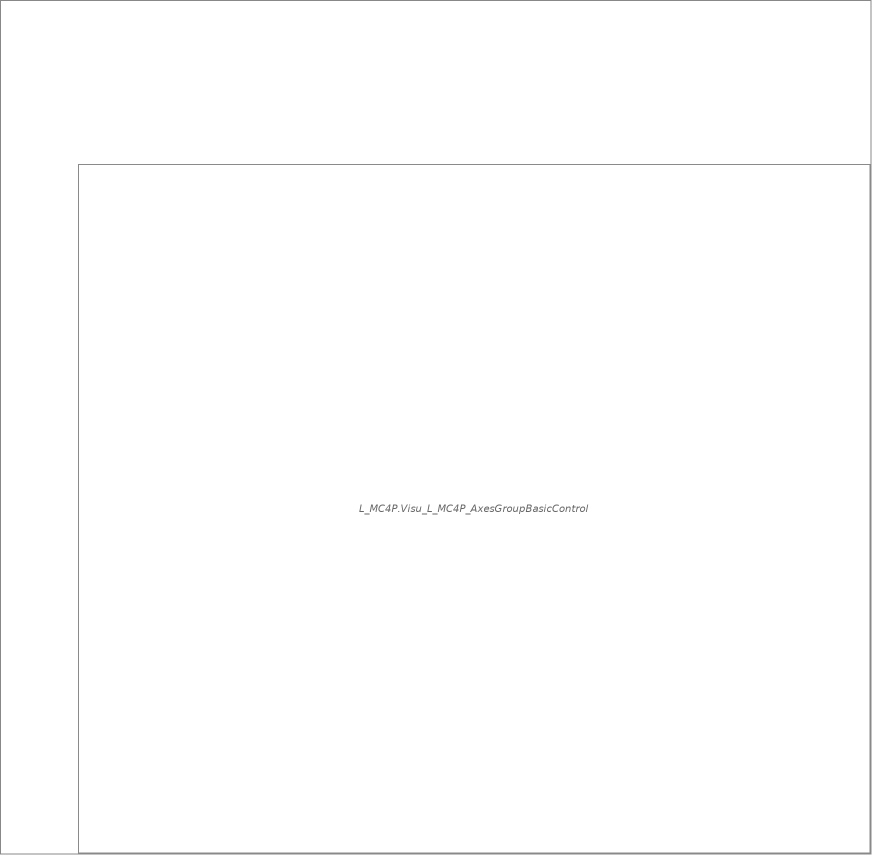
VISUALIZATION ABControl  // 872x855
    Frame (78,164 792x689)
        shows L_MC4P.Visu_L_MC4P_AxesGroupBasicControl(m_Input_FB := AGBControl)
END_VISUALIZATION

// Controller_3200C/Application/B5_VISUAL/Products
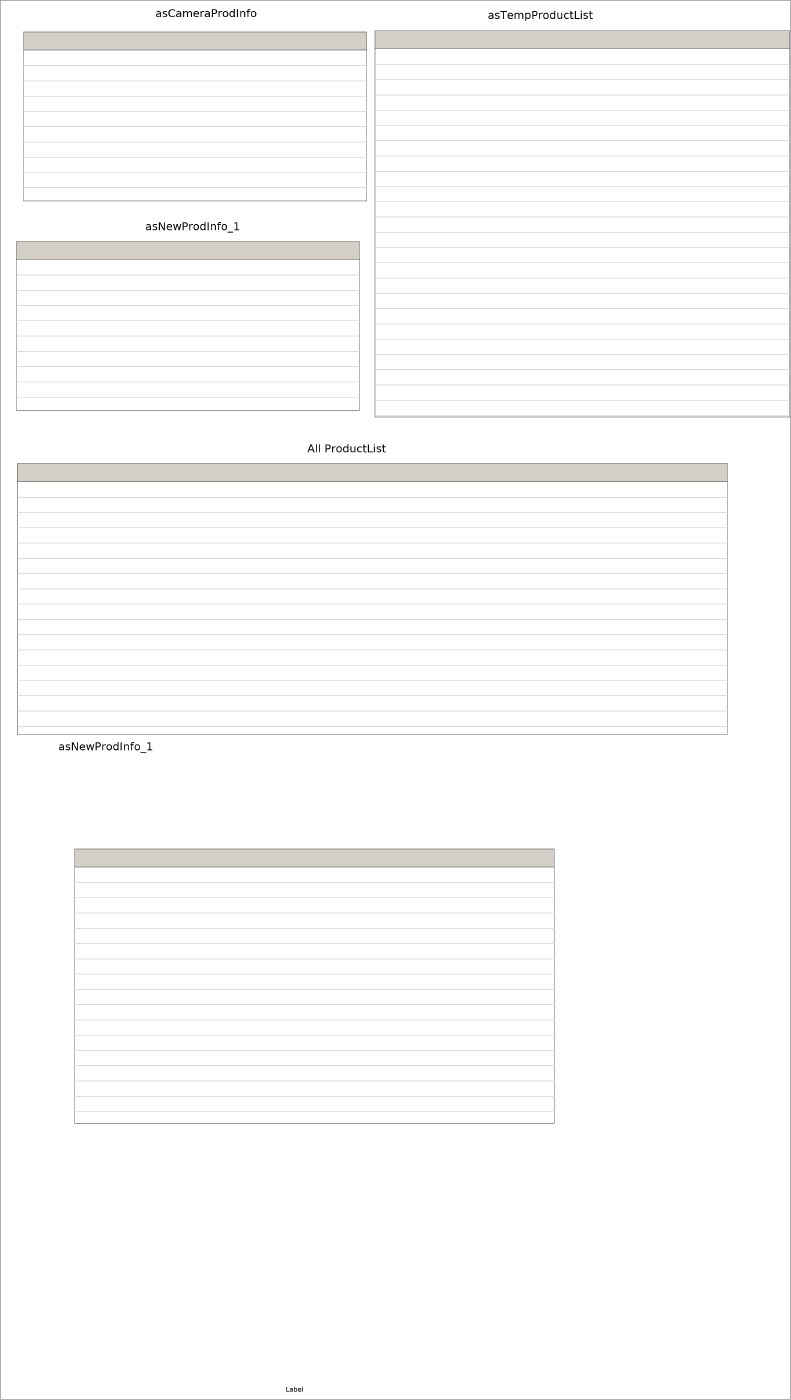
VISUALIZATION Products  // 1296x2293
    Label (225,7 226x30), "asCameraProdInfo"
    Table (28,759 1164x444), data array: Main.BufferHandling.asAllProductListInfo
        p3726181087: CameraProduct[INDEX].lrPosition
        p3136911649: CameraProduct[INDEX].lrLockedInfeedPos
        p3854506369: Main.BufferHandling.asAllProductListInfo[INDEX].iAttribute
        p1892666644: Main.BufferHandling.asAllProductListInfo[INDEX].lrCameraPosX
        p338671338: Main.BufferHandling.asAllProductListInfo[INDEX].lrCameraPosY
        p2170511999: Main.BufferHandling.asAllProductListInfo[INDEX].lrCameraPosAuxC
        p3723444502: Main.BufferHandling.asAllProductListInfo[INDEX].lrPosAuxC
        p1218418051: Main.BufferHandling.asAllProductListInfo[INDEX].lrDeltaX
        p746581629: Main.BufferHandling.asAllProductListInfo[INDEX].lrDeltaY
        p3104783080: Main.BufferHandling.asAllProductListInfo[INDEX].lrLockedInfeedPos
        p2501879983: Main.BufferHandling.asAllProductListInfo[INDEX].lrPosition
        p4092479075: CameraAuxC
    Label (493,720 150x30), "All ProductList"
    Label (780,10 211x30), "asTempProductList"
    Label (68,1208 211x30), "asNewProdInfo_1"
    Table (614,50 680x633), data array: Main.LoadDistribution.asTempProductList
        p3726181087: CameraProduct[INDEX].lrPosition
        p3136911649: CameraProduct[INDEX].lrLockedInfeedPos
        p3854506369: Main.LoadDistribution.asTempProductList[INDEX].iAttribute
        p1892666644: Main.LoadDistribution.asTempProductList[INDEX].lrCameraPosX
        p338671338: Main.LoadDistribution.asTempProductList[INDEX].lrCameraPosY
        p2170511999: Main.LoadDistribution.asTempProductList[INDEX].lrCameraPosAuxC
        p3723444502: Main.LoadDistribution.asTempProductList[INDEX].lrPosAuxC
        p1218418051: Main.LoadDistribution.asTempProductList[INDEX].lrDeltaX
        p746581629: Main.LoadDistribution.asTempProductList[INDEX].lrDeltaY
        p3104783080: Main.LoadDistribution.asTempProductList[INDEX].lrLockedInfeedPos
        p2501879983: Main.LoadDistribution.asTempProductList[INDEX].lrPosition
        p7306298: Main.LoadDistribution.asTempProductList[INDEX].iRank
    Table (38,52 563x277), data array: Main.LoadDistribution.asCameraProdInfo
        p3726181087: CameraProduct[INDEX].lrPosition
        p3136911649: CameraProduct[INDEX].lrLockedInfeedPos
        p3854506369: Main.LoadDistribution.asCameraProdInfo[INDEX].iAttribute
        p1892666644: Main.LoadDistribution.asCameraProdInfo[INDEX].lrCameraPosX
        p338671338: Main.LoadDistribution.asCameraProdInfo[INDEX].lrCameraPosY
        p2170511999: Main.LoadDistribution.asCameraProdInfo[INDEX].lrCameraPosAuxC
        p3723444502: Main.LoadDistribution.asCameraProdInfo[INDEX].lrPosAuxC
        p1218418051: Main.LoadDistribution.asCameraProdInfo[INDEX].lrDeltaX
        p746581629: Main.LoadDistribution.asCameraProdInfo[INDEX].lrDeltaY
        p3104783080: Main.LoadDistribution.asCameraProdInfo[INDEX].lrLockedInfeedPos
        p2501879983: Main.LoadDistribution.asCameraProdInfo[INDEX].lrPosition
    Table (26,395 563x277), data array: Main.LoadDistribution.asNewProdInfo_1
        p3726181087: CameraProduct[INDEX].lrPosition
        p3136911649: CameraProduct[INDEX].lrLockedInfeedPos
        p3854506369: Main.LoadDistribution.asNewProdInfo_1[INDEX].iAttribute
        p1892666644: Main.LoadDistribution.asNewProdInfo_1[INDEX].lrCameraPosX
        p338671338: Main.LoadDistribution.asNewProdInfo_1[INDEX].lrCameraPosY
        p2170511999: Main.LoadDistribution.asNewProdInfo_1[INDEX].lrCameraPosAuxC
        p3723444502: Main.LoadDistribution.asNewProdInfo_1[INDEX].lrPosAuxC
        p1218418051: Main.LoadDistribution.asNewProdInfo_1[INDEX].lrDeltaX
        p746581629: Main.LoadDistribution.asNewProdInfo_1[INDEX].lrDeltaY
        p3104783080: Main.LoadDistribution.asNewProdInfo_1[INDEX].lrLockedInfeedPos
        p2501879983: Main.LoadDistribution.asNewProdInfo_1[INDEX].lrPosition
        p7306298: Main.LoadDistribution.asNewProdInfo_1[INDEX].iRank
    Label (203,356 226x30), "asNewProdInfo_1"
    Label (408,2261 150x30), "Label"
    Table (122,1390 786x450), data array: CustomerPrgHandling.BoxBuffer.asAllProductListInfo
        p3854506369: CustomerPrgHandling.BoxBuffer.asAllProductListInfo[INDEX].iAttribute
        p1892666644: CustomerPrgHandling.BoxBuffer.asAllProductListInfo[INDEX].lrDetectPosX
        p338671338: CustomerPrgHandling.BoxBuffer.asAllProductListInfo[INDEX].lrDetectPosY
        p2170511999: CustomerPrgHandling.BoxBuffer.asAllProductListInfo[INDEX].lrDetectPosAuxC
        p3723444502: CustomerPrgHandling.BoxBuffer.asAllProductListInfo[INDEX].lrDeltaX
        p1218418051: CustomerPrgHandling.BoxBuffer.asAllProductListInfo[INDEX].lrDeltaY
        p746581629: CustomerPrgHandling.BoxBuffer.asAllProductListInfo[INDEX].lrPosAuxC
        p3104783080: CustomerPrgHandling.BoxBuffer.asAllProductListInfo[INDEX].lrLockedOutfeedPos
        p2501879983: CustomerPrgHandling.BoxBuffer.asAllProductListInfo[INDEX].lrPosition
END_VISUALIZATION

// Controller_3200C/Application/B5_VISUAL/SensorBuffer
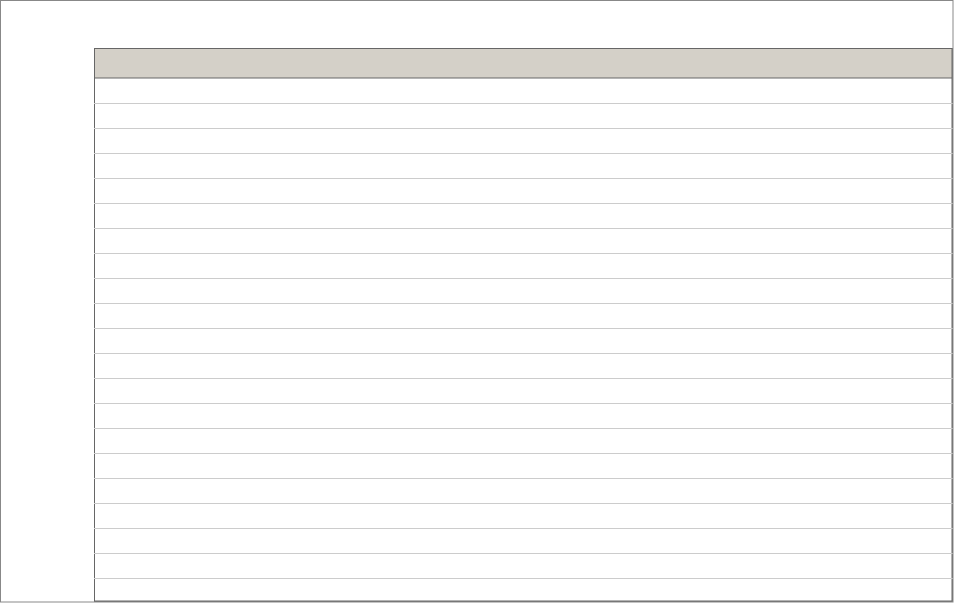
VISUALIZATION SensorBuffer  // 954x603
R_IN_OUT
	
END_VAR
    Table (94,48 858x553), data array: Main.SensorBufferHandler.asAllProductListInfo
        p3854506369: Main.SensorBufferHandler.asAllProductListInfo[INDEX].lrDetectPosX
        p1892666644: Main.SensorBufferHandler.asAllProductListInfo[INDEX].lrDetectPosY
        p338671338: Main.SensorBufferHandler.asAllProductListInfo[INDEX].lrDetectPosAuxC
        p2170511999: Main.SensorBufferHandler.asAllProductListInfo[INDEX].lrDeltaX
        p3723444502: Main.SensorBufferHandler.asAllProductListInfo[INDEX].lrDeltaY
        p1218418051: Main.SensorBufferHandler.asAllProductListInfo[INDEX].lrPosAuxC
        p746581629: Main.SensorBufferHandler.asAllProductListInfo[INDEX].lrLockedOutfeedPos
        p3104783080: Main.SensorBufferHandler.asAllProductListInfo[INDEX].lrPosition
END_VISUALIZATION

// Controller_3200C/Application/B5_VISUAL/MultiPick
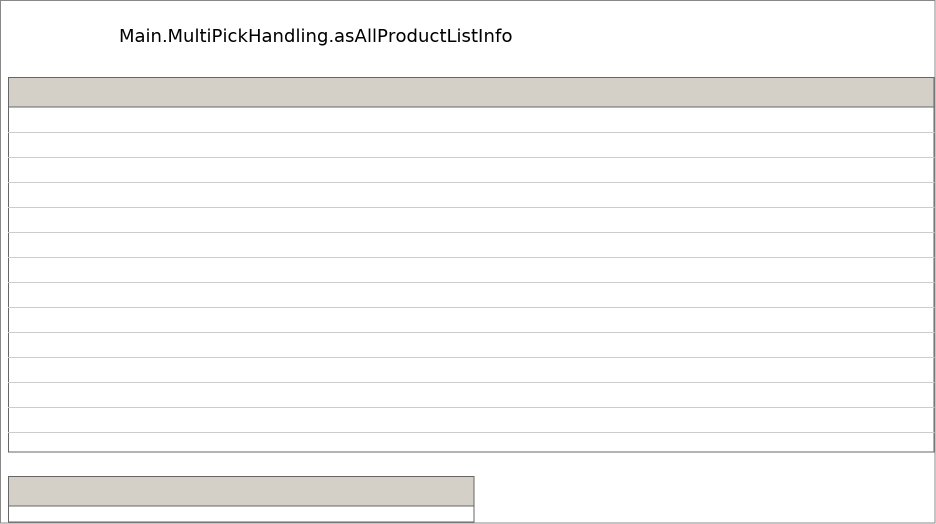
VISUALIZATION MultiPick  // 936x524
    Label (88,21 456x30), "Main.MultiPickHandling.asAllProductListInfo"
    Table (8,77 926x375), data array: Main.MultiPickHandling.asAllProductListInfo
        p3854506369: Main.MultiPickHandling.asAllProductListInfo[INDEX].iAttribute
        p2170511999: Main.MultiPickHandling.asAllProductListInfo[INDEX].lrCameraPosAuxC
        p3723444502: Main.MultiPickHandling.asAllProductListInfo[INDEX].lrPosAuxC
        p1218418051: Main.MultiPickHandling.asAllProductListInfo[INDEX].lrDeltaX
        p746581629: Main.MultiPickHandling.asAllProductListInfo[INDEX].lrDeltaY
        p3104783080: Main.MultiPickHandling.asAllProductListInfo[INDEX].lrLockedInfeedPos
        p2501879983: Main.MultiPickHandling.asAllProductListInfo[INDEX].lrPosition
        p1755163831: CameraPosY
        p338671338: Main.MultiPickHandling.asAllProductListInfo[INDEX].lrCameraPosY
        p511219082: CameraPosX
        p1892666644: Main.MultiPickHandling.asAllProductListInfo[INDEX].lrCameraPosX
    Table (8,476 466x46), data array: Main.MultiPickHandling.iNrOfProductsOnTrack
        p3854506369: Main.MultiPickHandling.iNrOfProductsOnTrack
        p1892666644: Main.MultiPickHandling.asAllProductListInfo[INDEX].lrCameraPosX
        p338671338: Main.MultiPickHandling.asAllProductListInfo[INDEX].lrCameraPosY
        p2170511999: Main.MultiPickHandling.asAllProductListInfo[INDEX].lrCameraPosAuxC
        p3723444502: Main.MultiPickHandling.asAllProductListInfo[INDEX].lrPosAuxC
        p1218418051: Main.MultiPickHandling.asAllProductListInfo[INDEX].lrDeltaX
        p746581629: Main.MultiPickHandling.asAllProductListInfo[INDEX].lrDeltaY
        p3104783080: Main.MultiPickHandling.asAllProductListInfo[INDEX].lrLockedInfeedPos
        p2501879983: Main.MultiPickHandling.asAllProductListInfo[INDEX].lrPosition
END_VISUALIZATION
